{attribute 'pack_mode' := '1'}
TYPE HomeAxis EXTENDS IncomingMessage :
STRUCT
	axisIndex: INT; (* 1 or 2.*)
END_STRUCT
END_TYPE

(* stored: Version 1.1.0.1, ProductVersion 3.1.4022.12
   DUT HomeAxis: Id {147fce52-b8c3-410d-ac5c-9f50ecb38028} *)
